PROGRAM MAIN
VAR
END_VAR

END_PROGRAM

(* stored: Version 1.1.0.1
   POU MAIN: Id {a8605b09-14c1-42af-ad44-9e0837ea999a} *)
